{attribute 'pack_mode' := '1'}
TYPE U_Debug_ST_3102 :
UNION
	Bytes	:ARRAY[0..499] OF BYTE;
	st3102	:ST_3102_Navitrol_status;
END_UNION
END_TYPE

(* stored: Version 1.1.0.1, ProductVersion 3.1.4026.17
   DUT U_Debug_ST_3102: Id {aa552a03-7f56-43af-a6ae-450becec7a51} *)
